% RSLogix 500 project CONVEYOR DIGITAL CONTROL_BAK048.RSS, saved by version 8.30.00.16 %
PROJECT "UNTITLED"    % processor: Bul.1763 MicroLogix 1100 Series B %

PROGRAM FILES
  LAD 2 "MAIN"  3 rungs
  LAD 3 "DIGITAL IO"  9 rungs
  LAD 4 "CONTROLS"  13 rungs
  LAD 5 "ALARMS"  2 rungs

DATA FILES
  O0 OUTPUT  4 elements
  I1 INPUT  6 elements
  S2 STATUS  66 elements
  B3 BINARY  5 elements
  T4 TIMER  1 elements
  C5 COUNTER  1 elements
  R6 CONTROL  1 elements
  N7 INTEGER  1 elements
  F8 FLOAT  1 elements

LADDER 2 "MAIN"
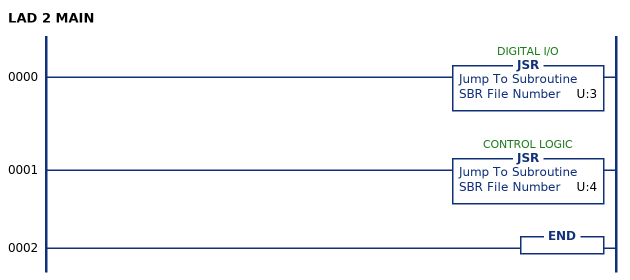
% Rung: 0 %
SOR JSR U:3 EOR
%   U:3  "DIGITAL I/O" %
% Rung: 1 %
SOR JSR U:4 EOR
%   U:4  "CONTROL LOGIC" %
% Rung: 2 %
SOR END EOR

LADDER 3 "DIGITAL IO"
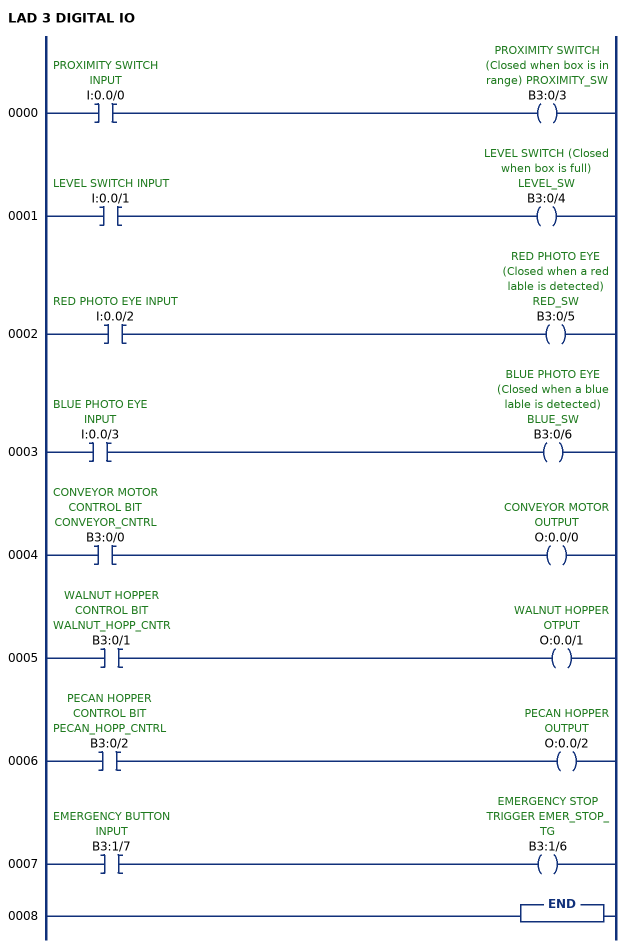
% Rung: 0 %
SOR XIC I:0.0/0 OTE B3:0/3 EOR
%   I:0.0/0  "PROXIMITY SWITCH INPUT" %
%   B3:0/3  PROXIMITY_SW  "PROXIMITY SWITCH (Closed when box is in range)" %
% Rung: 1 %
SOR XIC I:0.0/1 OTE B3:0/4 EOR
%   I:0.0/1  "LEVEL SWITCH INPUT" %
%   B3:0/4  LEVEL_SW  "LEVEL SWITCH (Closed when box is full)" %
% Rung: 2 %
SOR XIC I:0.0/2 OTE B3:0/5 EOR
%   I:0.0/2  "RED PHOTO EYE INPUT" %
%   B3:0/5  RED_SW  "RED PHOTO EYE (Closed when a red lable is detected)" %
% Rung: 3 %
SOR XIC I:0.0/3 OTE B3:0/6 EOR
%   I:0.0/3  "BLUE PHOTO EYE INPUT" %
%   B3:0/6  BLUE_SW  "BLUE PHOTO EYE (Closed when a blue lable is detected)" %
% Rung: 4 %
SOR XIC B3:0/0 OTE O:0.0/0 EOR
%   B3:0/0  CONVEYOR_CNTRL  "CONVEYOR MOTOR CONTROL BIT" %
%   O:0.0/0  "CONVEYOR MOTOR OUTPUT" %
% Rung: 5 %
SOR XIC B3:0/1 OTE O:0.0/1 EOR
%   B3:0/1  WALNUT_HOPP_CNTR  "WALNUT HOPPER CONTROL BIT" %
%   O:0.0/1  "WALNUT HOPPER OTPUT" %
% Rung: 6 %
SOR XIC B3:0/2 OTE O:0.0/2 EOR
%   B3:0/2  PECAN_HOPP_CNTRL  "PECAN HOPPER CONTROL BIT" %
%   O:0.0/2  "PECAN HOPPER OUTPUT" %
% Rung: 7 %
SOR XIC B3:1/7 OTE B3:1/6 EOR
%   B3:1/7  "EMERGENCY BUTTON INPUT" %
%   B3:1/6  EMER_STOP_TG  "EMERGENCY STOP TRIGGER" %
% Rung: 8 %
SOR END EOR

LADDER 4 "CONTROLS"
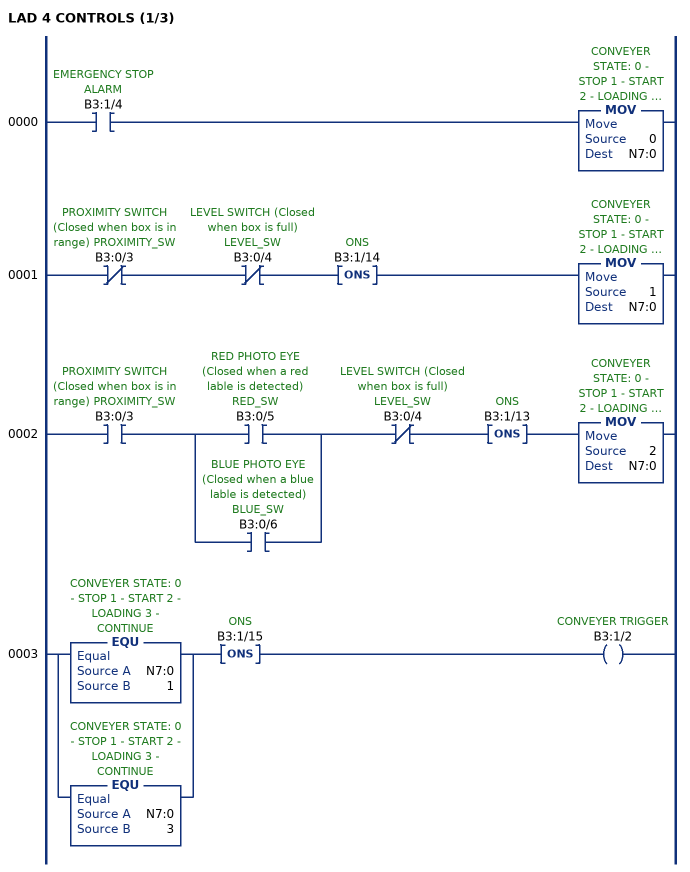
% Rung: 0 %
SOR XIC B3:1/4 MOV 0 N7:0 EOR
%   B3:1/4  "EMERGENCY STOP ALARM" %
%   N7:0  "CONVEYER STATE: 0 - STOP 1 - START 2 - LOADING 3 - CONTINUE" %
% Rung: 1 %
SOR XIO B3:0/3 XIO B3:0/4 ONS B3:1/14 MOV 1 N7:0 EOR
%   B3:0/3  PROXIMITY_SW  "PROXIMITY SWITCH (Closed when box is in range)" %
%   B3:0/4  LEVEL_SW  "LEVEL SWITCH (Closed when box is full)" %
%   B3:1/14  "ONS" %
%   N7:0  "CONVEYER STATE: 0 - STOP 1 - START 2 - LOADING 3 - CONTINUE" %
% Rung: 2 %
SOR XIC B3:0/3 BST XIC B3:0/5 NXB XIC B3:0/6 BND XIO B3:0/4 ONS B3:1/13 MOV 2 N7:0 EOR
%   B3:0/3  PROXIMITY_SW  "PROXIMITY SWITCH (Closed when box is in range)" %
%   B3:0/5  RED_SW  "RED PHOTO EYE (Closed when a red lable is detected)" %
%   B3:0/6  BLUE_SW  "BLUE PHOTO EYE (Closed when a blue lable is detected)" %
%   B3:0/4  LEVEL_SW  "LEVEL SWITCH (Closed when box is full)" %
%   B3:1/13  "ONS" %
%   N7:0  "CONVEYER STATE: 0 - STOP 1 - START 2 - LOADING 3 - CONTINUE" %
% Rung: 3 %
SOR BST EQU N7:0 1 NXB EQU N7:0 3 BND ONS B3:1/15 OTE B3:1/2 EOR
%   N7:0  "CONVEYER STATE: 0 - STOP 1 - START 2 - LOADING 3 - CONTINUE" %
%   B3:1/15  "ONS" %
%   B3:1/2  "CONVEYER TRIGGER" %

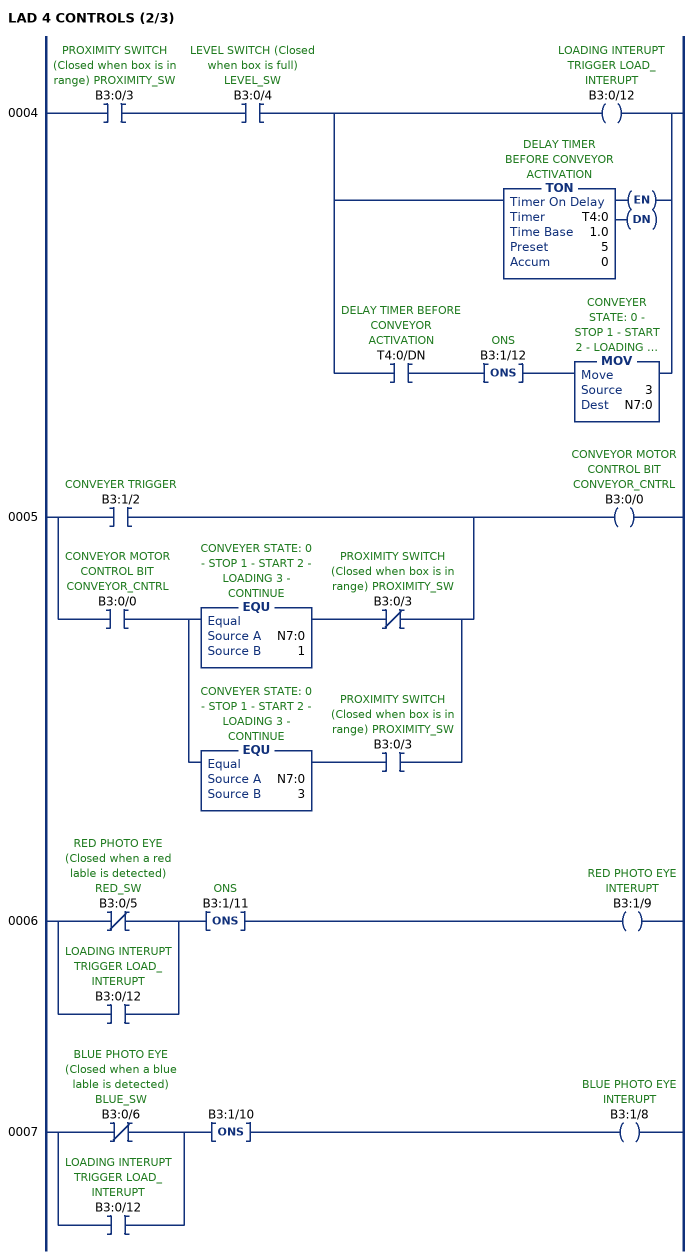
% Rung: 4 %
SOR XIC B3:0/3 XIC B3:0/4 BST OTE B3:0/12 NXB TON T4:0 1.0 5 0 NXB XIC T4:0/DN ONS B3:1/12 MOV 3 N7:0 BND EOR
%   B3:0/3  PROXIMITY_SW  "PROXIMITY SWITCH (Closed when box is in range)" %
%   B3:0/4  LEVEL_SW  "LEVEL SWITCH (Closed when box is full)" %
%   B3:0/12  LOAD_INTERUPT  "LOADING INTERUPT TRIGGER" %
%   T4:0  "DELAY TIMER BEFORE CONVEYOR ACTIVATION" %
%   B3:1/12  "ONS" %
%   N7:0  "CONVEYER STATE: 0 - STOP 1 - START 2 - LOADING 3 - CONTINUE" %
% Rung: 5 %
SOR BST XIC B3:1/2 NXB XIC B3:0/0 BST EQU N7:0 1 XIO B3:0/3 NXB EQU N7:0 3 XIC B3:0/3 BND BND OTE B3:0/0 EOR
%   B3:1/2  "CONVEYER TRIGGER" %
%   B3:0/0  CONVEYOR_CNTRL  "CONVEYOR MOTOR CONTROL BIT" %
%   N7:0  "CONVEYER STATE: 0 - STOP 1 - START 2 - LOADING 3 - CONTINUE" %
%   B3:0/3  PROXIMITY_SW  "PROXIMITY SWITCH (Closed when box is in range)" %
% Rung: 6 %
SOR BST XIO B3:0/5 NXB XIC B3:0/12 BND ONS B3:1/11 OTE B3:1/9 EOR
%   B3:0/5  RED_SW  "RED PHOTO EYE (Closed when a red lable is detected)" %
%   B3:0/12  LOAD_INTERUPT  "LOADING INTERUPT TRIGGER" %
%   B3:1/11  "ONS" %
%   B3:1/9  "RED PHOTO EYE INTERUPT" %
% Rung: 7 %
SOR BST XIO B3:0/6 NXB XIC B3:0/12 BND ONS B3:1/10 OTE B3:1/8 EOR
%   B3:0/6  BLUE_SW  "BLUE PHOTO EYE (Closed when a blue lable is detected)" %
%   B3:0/12  LOAD_INTERUPT  "LOADING INTERUPT TRIGGER" %
%   B3:1/8  "BLUE PHOTO EYE INTERUPT" %

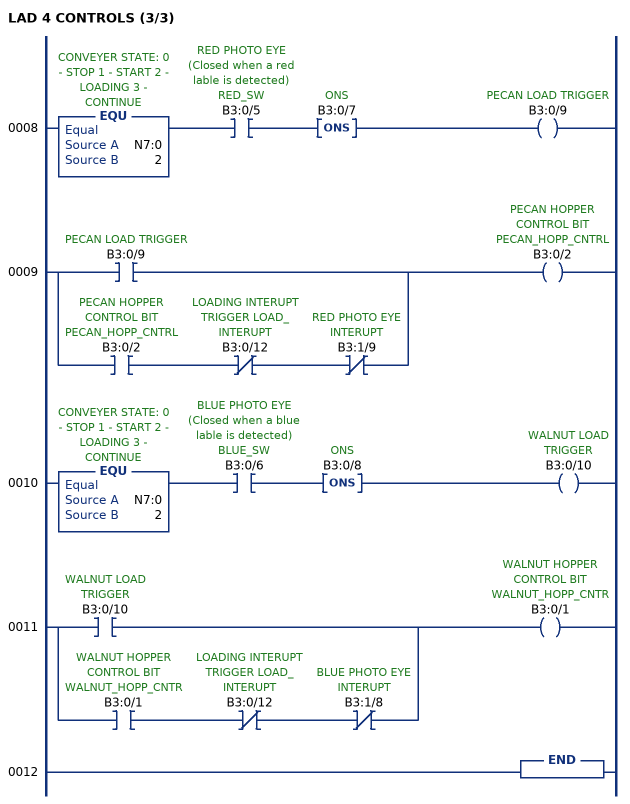
% Rung: 8 %
SOR EQU N7:0 2 XIC B3:0/5 ONS B3:0/7 OTE B3:0/9 EOR
%   N7:0  "CONVEYER STATE: 0 - STOP 1 - START 2 - LOADING 3 - CONTINUE" %
%   B3:0/5  RED_SW  "RED PHOTO EYE (Closed when a red lable is detected)" %
%   B3:0/7  "ONS" %
%   B3:0/9  "PECAN LOAD TRIGGER" %
% Rung: 9 %
SOR BST XIC B3:0/9 NXB XIC B3:0/2 XIO B3:0/12 XIO B3:1/9 BND OTE B3:0/2 EOR
%   B3:0/9  "PECAN LOAD TRIGGER" %
%   B3:0/2  PECAN_HOPP_CNTRL  "PECAN HOPPER CONTROL BIT" %
%   B3:0/12  LOAD_INTERUPT  "LOADING INTERUPT TRIGGER" %
%   B3:1/9  "RED PHOTO EYE INTERUPT" %
% Rung: 10 %
SOR EQU N7:0 2 XIC B3:0/6 ONS B3:0/8 OTE B3:0/10 EOR
%   N7:0  "CONVEYER STATE: 0 - STOP 1 - START 2 - LOADING 3 - CONTINUE" %
%   B3:0/6  BLUE_SW  "BLUE PHOTO EYE (Closed when a blue lable is detected)" %
%   B3:0/8  "ONS" %
%   B3:0/10  "WALNUT LOAD TRIGGER" %
% Rung: 11 %
SOR BST XIC B3:0/10 NXB XIC B3:0/1 XIO B3:0/12 XIO B3:1/8 BND OTE B3:0/1 EOR
%   B3:0/10  "WALNUT LOAD TRIGGER" %
%   B3:0/1  WALNUT_HOPP_CNTR  "WALNUT HOPPER CONTROL BIT" %
%   B3:0/12  LOAD_INTERUPT  "LOADING INTERUPT TRIGGER" %
%   B3:1/8  "BLUE PHOTO EYE INTERUPT" %
% Rung: 12 %
SOR END EOR

LADDER 5 "ALARMS"
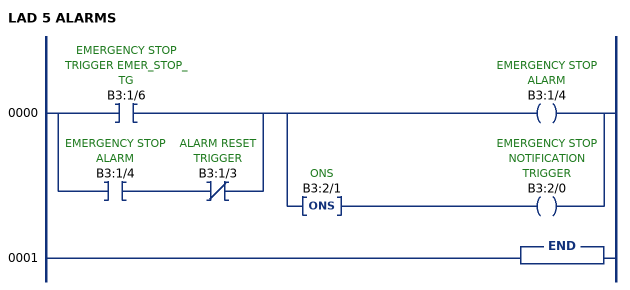
% Rung: 0 %
SOR BST XIC B3:1/6 NXB XIC B3:1/4 XIO B3:1/3 BND BST OTE B3:1/4 NXB ONS B3:2/1 OTE B3:2/0 BND EOR
%   B3:1/6  EMER_STOP_TG  "EMERGENCY STOP TRIGGER" %
%   B3:1/4  "EMERGENCY STOP ALARM" %
%   B3:1/3  "ALARM RESET TRIGGER" %
%   B3:2/1  "ONS" %
%   B3:2/0  "EMERGENCY STOP NOTIFICATION TRIGGER" %
% Rung: 1 %
SOR END EOR

OTHER DOCUMENTED ADDRESSES
  B3:0/11  "ONS"
  B3:0/13  "NEXT CYCLE FLAG"
  B3:0/14  "ONS"
  B3:0/15  "ONS"
  B3:1/0  "ONS"
  B3:1/1  "ONS"
  B3:1/5  "ONS"

DATA TABLE (non-zero values as saved)
DATA B3
% B3:0 % 0X4000 0X4002 0X0000 0X0000 0X0000
DATA T4
% .PRE .ACC %
% T4:0 % 5 0
DATA N7
% N7:0 % 1
